# EPICS substitutions: apps/iocBoot/ioctorusDaq/wf2root.substitutions
file "db/wf2root_ctrl.db" {
    pattern { P, R, PATH, PREFIX }
    { B_TORUS:, DAQ_REC:, "/logs/torus/", "torus_" }
}

file "db/wf2root_data.db" {
    pattern { P, R, WF, WF_FTVL, WF_NELM, WF_PV }
    { B_TORUS:, DAQ_REC:, VT1, FLOAT, 2000, hallb-crio-tor-fast:IOC:VT1 }
    { B_TORUS:, DAQ_REC:, VT2, FLOAT, 2000, hallb-crio-tor-fast:IOC:VT2 }
    { B_TORUS:, DAQ_REC:, VT3, FLOAT, 2000, hallb-crio-tor-fast:IOC:VT3 }
    { B_TORUS:, DAQ_REC:, VT4, FLOAT, 2000, hallb-crio-tor-fast:IOC:VT4 }
    { B_TORUS:, DAQ_REC:, VT5, FLOAT, 2000, hallb-crio-tor-fast:IOC:VT5 }
    { B_TORUS:, DAQ_REC:, VT6, FLOAT, 2000, hallb-crio-tor-fast:IOC:VT6 }
    { B_TORUS:, DAQ_REC:, VT7, FLOAT, 2000, hallb-crio-tor-fast:IOC:VT7 }
    { B_TORUS:, DAQ_REC:, VT8, FLOAT, 2000, hallb-crio-tor-fast:IOC:VT8 }
    { B_TORUS:, DAQ_REC:, VT9, FLOAT, 2000, hallb-crio-tor-fast:IOC:VT9 }
    { B_TORUS:, DAQ_REC:, VT10, FLOAT, 2000, hallb-crio-tor-fast:IOC:VT10 }
    { B_TORUS:, DAQ_REC:, VT11, FLOAT, 2000, hallb-crio-tor-fast:IOC:VT11 }
    { B_TORUS:, DAQ_REC:, VT12, FLOAT, 2000, hallb-crio-tor-fast:IOC:VT12 }
    { B_TORUS:, DAQ_REC:, VT13, FLOAT, 2000, hallb-crio-tor-fast:IOC:VT13 }
    { B_TORUS:, DAQ_REC:, VT14, FLOAT, 2000, hallb-crio-tor-fast:IOC:VT14 }
    { B_TORUS:, DAQ_REC:, VT15, FLOAT, 2000, hallb-crio-tor-fast:IOC:VT15 }
    { B_TORUS:, DAQ_REC:, VT16, FLOAT, 2000, hallb-crio-tor-fast:IOC:VT16 }
    { B_TORUS:, DAQ_REC:, VT17, FLOAT, 2000, hallb-crio-tor-fast:IOC:VT17 }
    { B_TORUS:, DAQ_REC:, VT18, FLOAT, 2000, hallb-crio-tor-fast:IOC:VT18 }
    { B_TORUS:, DAQ_REC:, VT19, FLOAT, 2000, hallb-crio-tor-fast:IOC:VT19 }
    { B_TORUS:, DAQ_REC:, VT20, FLOAT, 2000, hallb-crio-tor-fast:IOC:VT20 }
    { B_TORUS:, DAQ_REC:, VT21, FLOAT, 2000, hallb-crio-tor-fast:IOC:VT21 }
    { B_TORUS:, DAQ_REC:, VT22, FLOAT, 2000, hallb-crio-tor-fast:IOC:VT22 }
    { B_TORUS:, DAQ_REC:, VT23, FLOAT, 2000, hallb-crio-tor-fast:IOC:VT23 }
    { B_TORUS:, DAQ_REC:, VT24, FLOAT, 2000, hallb-crio-tor-fast:IOC:VT24 }
    { B_TORUS:, DAQ_REC:, IDCCT1, FLOAT, 2000, hallb-crio-tor-fast:IOC:IDCCT1 }
}

#
# !!! TEST DATA !!!
#
#file "db/wf2root_test.db" {
#    pattern { P, R, WF, WF_FTVL, WF_NELM }
#    { B_TORUS:, DAQ:, VT1, FLOAT, 2000 }
#    { B_TORUS:, DAQ:, VT2, FLOAT, 2000 }
#    { B_TORUS:, DAQ:, VT3, FLOAT, 2000 }
#    { B_TORUS:, DAQ:, VT4, FLOAT, 2000 }
#    { B_TORUS:, DAQ:, VT5, FLOAT, 2000 }
#    { B_TORUS:, DAQ:, VT6, FLOAT, 2000 }
#    { B_TORUS:, DAQ:, VT7, FLOAT, 2000 }
#    { B_TORUS:, DAQ:, VT8, FLOAT, 2000 }
#    { B_TORUS:, DAQ:, VT9, FLOAT, 2000 }
#    { B_TORUS:, DAQ:, VT10, FLOAT, 2000 }
#    { B_TORUS:, DAQ:, VT11, FLOAT, 2000 }
#    { B_TORUS:, DAQ:, VT12, FLOAT, 2000 }
#    { B_TORUS:, DAQ:, VT13, FLOAT, 2000 }
#    { B_TORUS:, DAQ:, VT14, FLOAT, 2000 }
#    { B_TORUS:, DAQ:, VT15, FLOAT, 2000 }
#    { B_TORUS:, DAQ:, VT16, FLOAT, 2000 }
#    { B_TORUS:, DAQ:, VT17, FLOAT, 2000 }
#    { B_TORUS:, DAQ:, VT18, FLOAT, 2000 }
#    { B_TORUS:, DAQ:, VT19, FLOAT, 2000 }
#    { B_TORUS:, DAQ:, VT20, FLOAT, 2000 }
#    { B_TORUS:, DAQ:, VT21, FLOAT, 2000 }
#    { B_TORUS:, DAQ:, VT22, FLOAT, 2000 }
#    { B_TORUS:, DAQ:, VT23, FLOAT, 2000 }
#}
